# EPICS autosave request: CARS/iocBoot/iocDCM/XFM_mono_params.req
# FILE... XFM_mono_params.req
$(P)$(M).VAL
